// TIA Portal V16 export
// export: Created 2022-11-14T17:35:53.9259262Z, ExportSetting WithDefaults, DisplayName Totally Integrated Automation Portal, DisplayVersion V16, DisplayName TIA Portal Version Control Interface, DisplayVersion V16, DisplayName TIA Portal Openness, DisplayVersion V16, DisplayName STEP 7 Professional, DisplayVersion V16, DisplayName STEP 7 Safety, DisplayVersion V16, DisplayName WinCC Advanced, DisplayVersion V16
TYPE "M20"
// stored: IsFailsafeCompliant false
   STRUCT
      M20_P00 : Int;   // Tipo di prestiro
      M20_P01 : Int;   // Coefficiente proporzionale per il regolatore PID
      M20_P02 : Int;   // Coefficiente integrale (Fase1 e Fase2) per il regolatore PID
      M20_P03 : Int;   // Coefficiente derivativo per il regolatore PID
      M20_P04 : Int;   // Coefficiente integrale (Fase3 e Fase4) per il regolatore PID
      M20_P05 : Int;   // Rampa di accelerazione per il tiro durante la Fase1
      M20_P06 : Int;   // Limite componente integrale nel transitorio dalla Fase2 alla Fase3
      M20_P07 : Int;   // Limite componente integrale nel transitorio dalla Fase3 alla Fase4
      M20_P08 : Int;   // Valore minimo ingresso analogico
      M20_P09 : Int;   // Valore massimo ingresso analogico
      M20_P10 : Int;   // Prestiro naturale dovuto al rapporto di riduzione
      M20_P11 : Int;   // Velocità per il jog in manuale dei rulli di prestiro
      M20_P12 : Int;   // Offset del rullo lento 10 equivale a 0
      M20_P13 : Int;   // Jog di velocità durante la partenza del braccio
      M20_P14 : Int;   // Tiro minimo durante la Fase4 di arresto e durante un arresto repentino
      M20_P15 : Int;   // Tempo (in decimi di secondo) dopo il quale i rulli si fermano per rottura film
      M20_P20 : Int;   // Velocità indicata da plc per la rotazione braccio e il carrello top
      M20_P21 : Int;   // Velocità indicata da plc per il carrello di prestiro e il trasporto di centro macchina
      M20_P22 : Int;   // Tiro indicato da plc
      M20_P23 : Int;   // Prestiro indicato da plc
      M20_P24 : Int;   // Valore di ingresso analogico AI0
      M20_P25 : Int;   // Tiro richiesto da plc compreso fra 0 e 100
   END_STRUCT;
END_TYPE
